DEVICE_TYPE GenericFORTE (* generic FORTE controller *)
  (* Standard: 61499 ITA; Description: Remotely Managed Device *)
  (* Version 1.0, 2016-09-20, Monika Wenger, fortiss GmbH, Initial version *)
  VAR_INPUT
    MGR_ID : WSTRING := "localhost:61499"; (* Device manager socket ID *)
  END_VAR
END_DEVICE_TYPE
